ADAPTER LREAL_EVENT (* Adapter Interface *)
  (* Standard: 61499-1 *)
  (* Version 0.0, 12/12/2023, Cheyan, Schneider Electric *)
  PACKAGE Main;
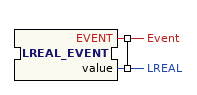
  EVENT_OUTPUT
    EVENT WITH value; (* Confirmation from Plug *)
  END_EVENT
  VAR_OUTPUT
    value : LREAL; (* Confirmation Data from Plug *)
  END_VAR
  SERVICE SOCKET/PLUG
    SEQUENCE request_confirm
      SOCKET.REQ(REQD) -> PLUG.REQ(REQD);
      PLUG.EVENT(value) -> SOCKET.EVENT(value);
    END_SEQUENCE
    SEQUENCE indication_response
      PLUG.IND(INDD) -> SOCKET.IND(INDD);
      SOCKET.RSP(RSPD) -> PLUG.RSP(RSPD);
    END_SEQUENCE
  END_SERVICE
END_ADAPTER
